PROGRAM F_FactoryIO_Write_Coils
VAR
	LFB_MBWriteCoils 	: FB_MBWriteCoils;
	bBusy: BOOL;
	bError: BOOL;

END_VAR

LFB_MBWriteCoils(
	sIPAddr := '127.0.0.1',
	nTCPPort := 505,
	nUnitID := 255,
	nQuantity := 16,
	nMBAddr := 0,
	cbLength := SIZEOF(GAB_FactoryIO_Outputs),
	pSrcAddr:= ADR(GAB_FactoryIO_Outputs), 
	bExecute := TRUE,
	tTimeout := T#1S,
	bBusy=> bBusy, 
	bError=> bError, 
	nErrId=>
);
LFB_MBWriteCoils(bExecute := FALSE);

END_PROGRAM

(* stored: Version 1.1.0.1, ProductVersion 3.1.4024.11
   POU F_FactoryIO_Write_Coils: Id {d4a8b314-3752-4f28-b57a-84f6b4497dd4}, SpecialFunc None *)
